FUNCTION TFNumeroPacchiSuLinea_OLD : UINT
VAR_INPUT
	HandlingPackTable : POINTER TO TFHandlingPackTable;
END_VAR
VAR
	i : UINT;
END_VAR

TFNumeroPacchiSuLinea := 0; 

FOR i:= 1 TO MAXHANDLINGPACK DO
	IF HandlingPackTable^.Table[i,1].PP THEN
		TFNumeroPacchiSuLinea := TFNumeroPacchiSuLinea +1;
	END_IF
END_FOR

END_FUNCTION

(* stored: Version 1.1.0.1, ProductVersion 3.1.4024.11
   POU TFNumeroPacchiSuLinea_OLD: Id {f3c3226b-56a9-4f5a-aff4-869969f77d4b}, SpecialFunc None *)
